{attribute 'GeneratedUsingTerminal: ER7041-0002-0024'}
{attribute addProperty BoxType "ER7041-0002-0024"}
{attribute addProperty Id "ControlAT %Q*Control_5FD4673D4"}
{attribute addProperty CRC "3125601106"}
{attribute addProperty Size "4"}
TYPE STM_Control_BA4CE352 :
STRUCT
	{attribute addProperty Name "Control"}
	Control AT %Q* : Control_5FD4673D;
END_STRUCT
END_TYPE

(* stored: Version 1.2.0.0, ProductVersion 3.1.4024.9
   DUT STM_Control_BA4CE352: Id {c490b4ad-ab79-429b-827e-8df787d0a340} *)
